FUNCTION_BLOCK FB_Blinker
VAR_INPUT
	tBlink						: TIME;					//脉冲宽度
END_VAR

VAR_OUTPUT
	bBlink						: BOOL;					//输出脉冲
	brBlink						: BOOL;					//输出脉冲上升沿
	bfBlink						: BOOL;					//输出脉冲上升沿
END_VAR

VAR
	{attribute 'hide'}
	tonBlink					: TON;					//计时
	{attribute 'hide'}
	rtBlink						: R_TRIG;				//脉冲上升沿
	{attribute 'hide'}
	ftBlink						: F_TRIG;				//脉冲下降沿
END_VAR

tonBlink(
	IN:=NOT tonBlink.Q,
	PT:=tBlink / 2,
	Q=>);
IF tonBlink.Q THEN
	bBlink:=NOT bBlink;
END_IF

rtBlink(CLK:=bBlink, Q=>brBlink);
ftBlink(CLK:=bBlink, Q=>bfBlink);

END_FUNCTION_BLOCK

(* stored: Version 1.1.0.1, ProductVersion 3.1.4024.9
   POU FB_Blinker: Id {af2dfb15-ef1c-4ed4-acf7-63a146640b48}, SpecialFunc None *)
